{attribute 'monitoring' := 'call'}
PROPERTY PUBLIC BT : TIME
GET
IF ton.IN
	AND NOT ton.Q
THEN
	BT 														:= ton.PT - ton.ET;
ELSE       													
	BT 														:= T#0MS;
END_IF
END_GET
END_PROPERTY

METHOD PUBLIC reset : BOOL //Return value = TRUE if execution finished
VAR_INPUT
END_VAR
Q 															:= FALSE;
TON(IN := FALSE);
reset													:= TRUE;
END_METHOD

END_FUNCTION_BLOCK

// POUs/TimeHelper/VeloLinearMeasurement
{attribute 'no_check'}
//Accumulates the covered distance based on the velocity input and the time IN is TRUE - used to detect jamped pieces on a conveyor
FUNCTION_BLOCK VeloLinearMeasurement
VAR_INPUT
	Enable													:	BOOL;	//Enable function (e.g. Conveyor on)
	ResetTrig												:	BOOL;	//Reset Q
	IN														:	BOOL; 	//Sensor input
	Velo													:	LREAL;  //mm/ms | m/s with FACTOR=1, m/min with FACTOR=16.666666666666668
	Factor													:	LREAL := 1.0;	//Used to convert "VELO" into mm/ms (e.g. 16.666666666666668 to convert m/min into mm/ms
END_VAR             										
VAR_OUTPUT          										
	Q														:	LREAL;	//Accumulated value in mm
END_VAR             										
VAR                 										
	tx														:	DWORD;
	last 													: 	DWORD;
	ms														: 	DWORD;
	mmProms													:	LREAL;
END_VAR


(* Get mm pro ms *)
mmProms 													:= VELO * FACTOR; 

(* read system time *)
tx 															:= TIME_TO_DWORD(TIME());

(* Sequence *)
IF ResetTrig THEN
	reset();
ELSIF IN AND Enable THEN
	(* add the current milliseconds *)
	ms 														:= (tx - last) + ms;
	Q 														:= ms * mmProms;
ELSE
	;
END_IF

(* Save last Cylcetime *)
last 														:= tx;

(**********************************************************************)

METHOD PUBLIC reset : bool //Return value = TRUE if execution finished
VAR_INPUT
END_VAR
Q 															:= 0;
ms 															:= 0;
reset													:= TRUE;
END_METHOD

END_FUNCTION_BLOCK

// Version/disclaimerStatement
// .. Disclaimer:: This function contains statements about the use of this library 
{attribute 'no-analysis'}
{attribute 'no_check'}
FUNCTION disclaimerStatement : WSTRING(1500)
VAR_INPUT
END_VAR
VAR
END_VAR

DisclaimerStatement := 
	"This disclaimer contains statements about the use of this library.

		-The use of this version of the library is free of charge 
		-It is incumbent on the customer to check and decide whether the library and provided function is suitable for use his particular application
		-This library is provided 'AS IS' and neither a part of TwinCAT3 nor directly supported by Beckhoff Automation
		-The use of the Library is at the Customer's own risk
		-There is no warranty given that the library and source code, which is made available with this library is complete or accurate
		-In no event will the author or Beckhoff Automation be liable for any claims, damages or other liability for errors and/or omissions arising from the use of the library
		-There is no right to expect maintenance, support, enhancements or modifications of the library as well as for updates or compatibility to updates of the library or TwinCAT3 if released
		
	For feedback or questions please contact the Beckhoff Industry Management for Electronics Manufacturing, D.Schlingmann@Beckhoff.com
	
	© Beckhoff Automation GmbH & Co. KG,
	The reproduction, distribution and utilisation of this library or parts of it as well as the communication of its content to others without express authorisation is prohibited held liable for the payment of damages.
	
	All rights reserved in the event of the grant of a patent, utility model or design.";

END_FUNCTION
